// SIMATIC S7-200 project (STEP 7-Micro/WIN), CPU 222 REL 01.22

SYMBOL_TABLE USR1
Always_On        SM0.0
First_Scan_On    SM0.1
Mod_0_IO_2       SM8.2    // 与SM8.3联合表示I/O扩展模块的输入点数目
Mod_0_IO_3       SM8.3    // 与SM8.2联合表示I/O扩展模块的输入点数目
Mod_0_IO_Type    SM8.4    // 该位表示当前I/O扩展模块的类型，（0表示数字量扩展模，1表示模拟量扩展模块）
Mod_0_Present    SM8.7    // 当该位为0时表示有I/O扩展模块存在
Unfiltered_AIW0  AIW0     // 每个扫描周期获得外部模拟量输入值
Filtered_Output  AQW0     // 包括最近N个模拟量采样值的均值
Filtered_Value   VW12     // 包括模拟量输入的均值
END_SYMBOL_TABLE

ORGANIZATION_BLOCK MAIN:OB1
TITLE= 题目：
// 模拟量输入的处理
// ***概述***
// 本例描述了模拟量模块EM235 3AI/1AQ与CPU-212或CPU-214一起使用的一种探讨。本例
// 中模拟量输入值是给定采样次数的采样平均值，然后试验决定怎样设置输出。EM235配置成
// 正负10V。
// ***程序和注释***
// 本程序描述了模拟量模块EM235(3AI/1AQ)的功能，从AIW0中取输入值，为了增加稳定性而
// 求多次采样值的平均值，再依据计算出的平均值在AQW0中输出模拟电压。
// 模拟量模块经过测试可提供模块错误信息。如果第一个扩展模块不是模拟量模块，Q1.0接通
// 另外模拟量模块检查到的错误是电源出错，则将CPU上Q1.1接通。模拟量模块上有EXTF字样。
// 本程序中所用除法是简单的移位除法(用采用次数的2的方次)。因为移位只花费较短的扫描时
// 间，该数能从2变化到32768 
// 输入字是12位长。如果采样次数大于16(2的4次方),那么和的长度将大于一个字(16位).于是
// 需要用双字(32位)存储采样和。为把输入值加到采样和中，你应当把它转成双字。
// 当输入数为负数时，最高有效字增添1；若为正值，最高有效字增添0来校正输入值。
// 
// 
BEGIN
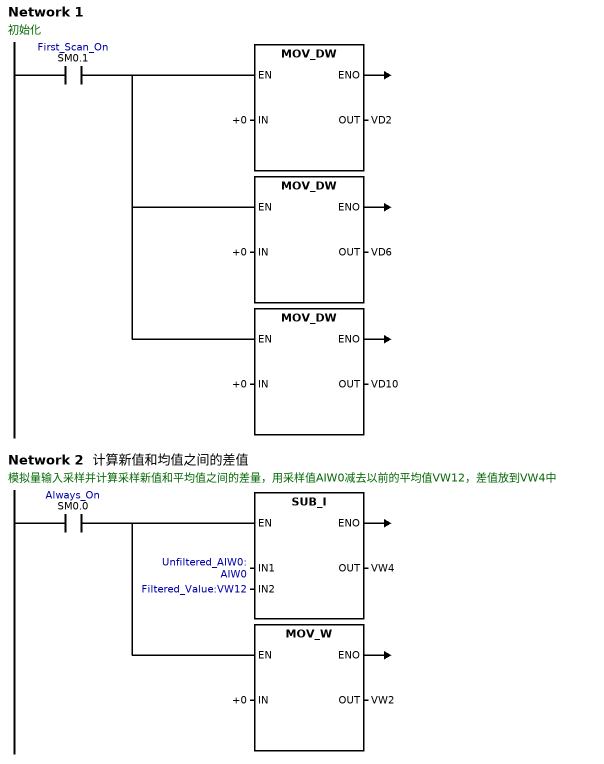
Network 1
// 初始化
// clear the working scratchpad area,
// clear the running sum,
// and clear the running average.
LD     First_Scan_On:SM0.1
MOVD   +0, VD2
MOVD   +0, VD6
MOVD   +0, VD10
Network 2 // 计算新值和均值之间的差值
// 模拟量输入采样并计算采样新值和平均值之间的差量，用采样值AIW0减去以前的平均值VW12，差值放到VW4中
// Every scan cycle,
// clear the most significant word
// of the working register,
// get the sampled AI value and
// put it in the scratchpad area,
// and compute the difference between
// the previous average and the new
// value and put the result in VW4.
LD     Always_On:SM0.0
MOVW   Unfiltered_AIW0:AIW0, VW4
-I     Filtered_Value:VW12, VW4
MOVW   +0, VW2
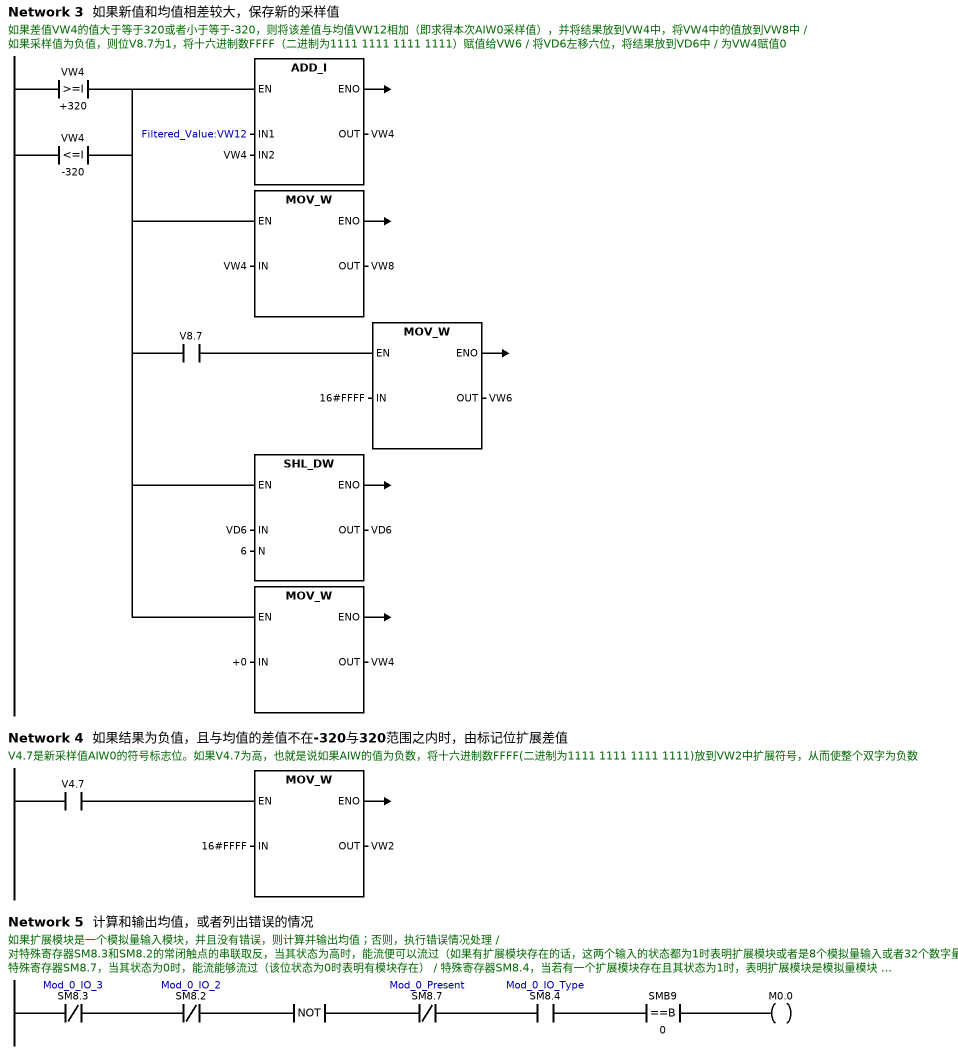
Network 3 // 如果新值和均值相差较大，保存新的采样值
// 如果差值VW4的值大于等于320或者小于等于-320，则将该差值与均值VW12相加（即求得本次AIW0采样值），并将结果放到VW4中，将VW4中的值放到VW8中
// 如果采样值为负值，则位V8.7为1，将十六进制数FFFF（二进制为1111 1111 1111 1111）赋值给VW6
// 将VD6左移六位，将结果放到VD6中
// 为VW4赋值0
// If the difference between the
// new value and the average
// value is greater than or equal
// to 320 counts,
// or if it is less than or equal
// to -320 counts,
// compute the last sample value
// without reading the analog
// input again
// and save the last sample.
// If the sample is negative,
// extend the sign to a double
// word value.
// Multiply this sample by the
// number of samples to produce
// a running sum.
// Zero the difference between
// the new value and the previous
// value.
LDW>=  VW4, +320
OW<=   VW4, -320
LPS
+I     Filtered_Value:VW12, VW4
MOVW   VW4, VW8
A      V8.7
MOVW   16#FFFF, VW6
LRD
SLD    VD6, 6
LPP
MOVW   +0, VW4
Network 4 // 如果结果为负值，且与均值的差值不在-320与320范围之内时，由标记位扩展差值
// V4.7是新采样值AIW0的符号标志位。如果V4.7为高，也就是说如果AIW的值为负数，将十六进制数FFFF(二进制为1111 1111 1111 1111)放到VW2中扩展符号，从而使整个双字为负数
// Read the sign bit to the new
// AI (WORD) value.
// If it is negative, extend the
// sign to make the entire DWORD
// negative.
LD     V4.7
MOVW   16#FFFF, VW2
Network 5 // 计算和输出均值，或者列出错误的情况
// 如果扩展模块是一个模拟量输入模块，并且没有错误，则计算并输出均值；否则，执行错误情况处理
// 对特殊寄存器SM8.3和SM8.2的常闭触点的串联取反，当其状态为高时，能流便可以流过（如果有扩展模块存在的话，这两个输入的状态都为1时表明扩展模块或者是8个模拟量输入或者32个数字量输出）
// 特殊寄存器SM8.7，当其状态为0时，能流能够流过（该位状态为0时表明有模块存在）
// 特殊寄存器SM8.4，当若有一个扩展模块存在且其状态为1时，表明扩展模块是模拟量模块
// 如果能流到了特殊位SMB9且其值为0，则说明该模拟量模块没有错误，计算并输出均值
// 将双字VD2的值加到VD6上来更新连续和值，将结果存放到VD6中
// 将VD6中的值右（和值）移6位获得连续均值，并将结果存放到VD10中
// 将VW12中的均值在AQW0中输出
// 任何前面的条件没有满足，如当前模块不是模拟量模块或者模块存在错误，则为AQW0赋值0来设定输出为错误值并且将Q0.0置位（在模拟量模块中有错误）来处理错误情况
// If an analog input module is
// present...
// and no module error is detected...
// update the running sum.
// Move the sum into the location
// for the running average,
// shift the DWORD right by 6 bits
// [ln(SampleSize)/ln(2)] bits,
// (same as SUM / SampleSize),
// and move the averaged value to
// the filtered output.
// If the module is not an analog
// module or a module error was
// detected,
// set the filtered output to
// the error value
// and set the AI Module Error bit.
LDN    Mod_0_IO_3:SM8.3
AN     Mod_0_IO_2:SM8.2
NOT
AN     Mod_0_Present:SM8.7
A      Mod_0_IO_Type:SM8.4
AB=    SMB9, 0
=      M0.0
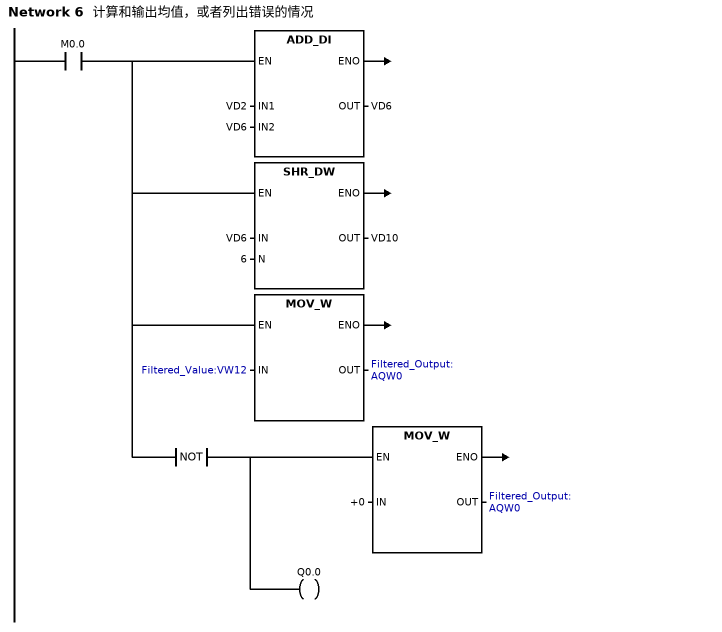
Network 6 // 计算和输出均值，或者列出错误的情况
// If an analog input module is
// present...
// and no module error is detected...
// update the running sum.
// Move the sum into the location
// for the running average,
// shift the DWORD right by 6 bits
// [ln(SampleSize)/ln(2)] bits,
// (same as SUM / SampleSize),
// and move the averaged value to
// the filtered output.
// If the module is not an analog
// module or a module error was
// detected,
// set the filtered output to
// the error value
// and set the AI Module Error bit.
// (network saved uncompiled; LAD cells follow)
// row 0: c0 -| |- M0.0 v  c1 --  c2 [ADD_DI EN:=power@row0, IN1:=VD2, IN2:=VD6, ENO=>power, OUT=>VD6]  c3 ->
// row 1: c0 ^v  c2 [box]
// row 2: c0 ^v  c1 --  c2 [SHR_DW EN:=power@row2, IN:=VD6, N:=6, ENO=>power, OUT=>VD10]  c3 ->
// row 3: c0 ^v  c2 [box]
// row 4: c0 ^v  c1 --  c2 [MOV_W EN:=power@row4, IN:=Filtered_Value:VW12, ENO=>power, OUT=>Filtered_Output:AQW0]  c3 ->
// row 5: c0 ^v  c2 [box]
// row 6: c0 ^  c1 -|NOT|-  v  c2 --  c3 [MOV_W EN:=power@row6, IN:=+0, ENO=>power, OUT=>Filtered_Output:AQW0]  c4 ->
// row 7: c1 ^v  c3 [box]
// row 8: c1 ^  c2 -( ) Q0.0
END_ORGANIZATION_BLOCK
